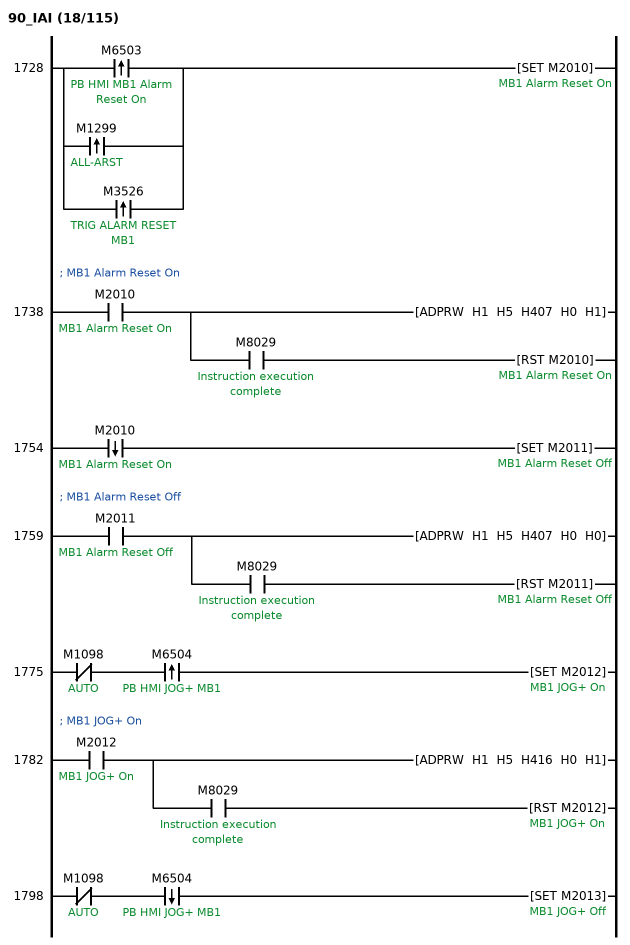
[picture p120: ladder of 90_IAI, rungs at steps 1728 to 1798]
1728  LDP     M6503  ; PB HMI MB1 Alarm Reset On
      ORP     M1299  ; ALL-ARST
      ORP     M3526  ; TRIG ALARM RESET MB1
      SET     M2010  ; MB1 Alarm Reset On
; MB1 Alarm Reset On
1738  LD      M2010  ; MB1 Alarm Reset On
      ADPRW   H1 H5 H407 H0 H1
      AND     M8029  ; Instruction execution complete
      RST     M2010  ; MB1 Alarm Reset On
1754  LDF     M2010  ; MB1 Alarm Reset On
      SET     M2011  ; MB1 Alarm Reset Off
; MB1 Alarm Reset Off
1759  LD      M2011  ; MB1 Alarm Reset Off
      ADPRW   H1 H5 H407 H0 H0
      AND     M8029  ; Instruction execution complete
      RST     M2011  ; MB1 Alarm Reset Off
1775  LDI     M1098  ; AUTO
      ANDP    M6504  ; PB HMI JOG+ MB1
      SET     M2012  ; MB1 JOG+ On
; MB1 JOG+ On
1782  LD      M2012  ; MB1 JOG+ On
      ADPRW   H1 H5 H416 H0 H1
      AND     M8029  ; Instruction execution complete
      RST     M2012  ; MB1 JOG+ On
1798  LDI     M1098  ; AUTO
      ANDF    M6504  ; PB HMI JOG+ MB1
      SET     M2013  ; MB1 JOG+ Off
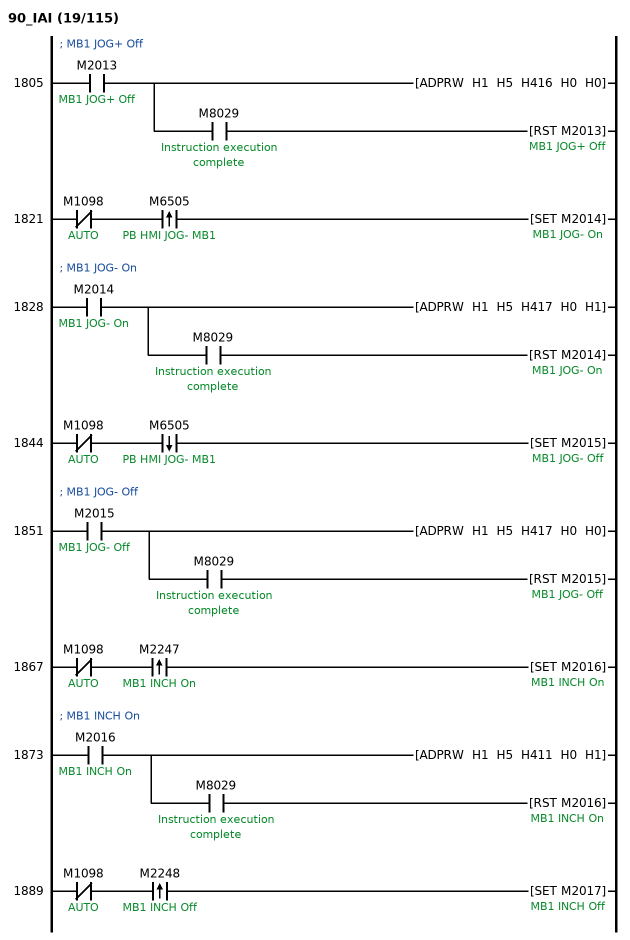
; MB1 JOG+ Off
1805  LD      M2013  ; MB1 JOG+ Off
      ADPRW   H1 H5 H416 H0 H0
      AND     M8029  ; Instruction execution complete
      RST     M2013  ; MB1 JOG+ Off
1821  LDI     M1098  ; AUTO
      ANDP    M6505  ; PB HMI JOG- MB1
      SET     M2014  ; MB1 JOG- On
; MB1 JOG- On
1828  LD      M2014  ; MB1 JOG- On
      ADPRW   H1 H5 H417 H0 H1
      AND     M8029  ; Instruction execution complete
      RST     M2014  ; MB1 JOG- On
1844  LDI     M1098  ; AUTO
      ANDF    M6505  ; PB HMI JOG- MB1
      SET     M2015  ; MB1 JOG- Off
; MB1 JOG- Off
1851  LD      M2015  ; MB1 JOG- Off
      ADPRW   H1 H5 H417 H0 H0
      AND     M8029  ; Instruction execution complete
      RST     M2015  ; MB1 JOG- Off
1867  LDI     M1098  ; AUTO
      ANDP    M2247  ; MB1 INCH On
      SET     M2016  ; MB1 INCH On
; MB1 INCH On
1873  LD      M2016  ; MB1 INCH On
      ADPRW   H1 H5 H411 H0 H1
      AND     M8029  ; Instruction execution complete
      RST     M2016  ; MB1 INCH On
1889  LDI     M1098  ; AUTO
      ANDP    M2248  ; MB1 INCH Off
      SET     M2017  ; MB1 INCH Off
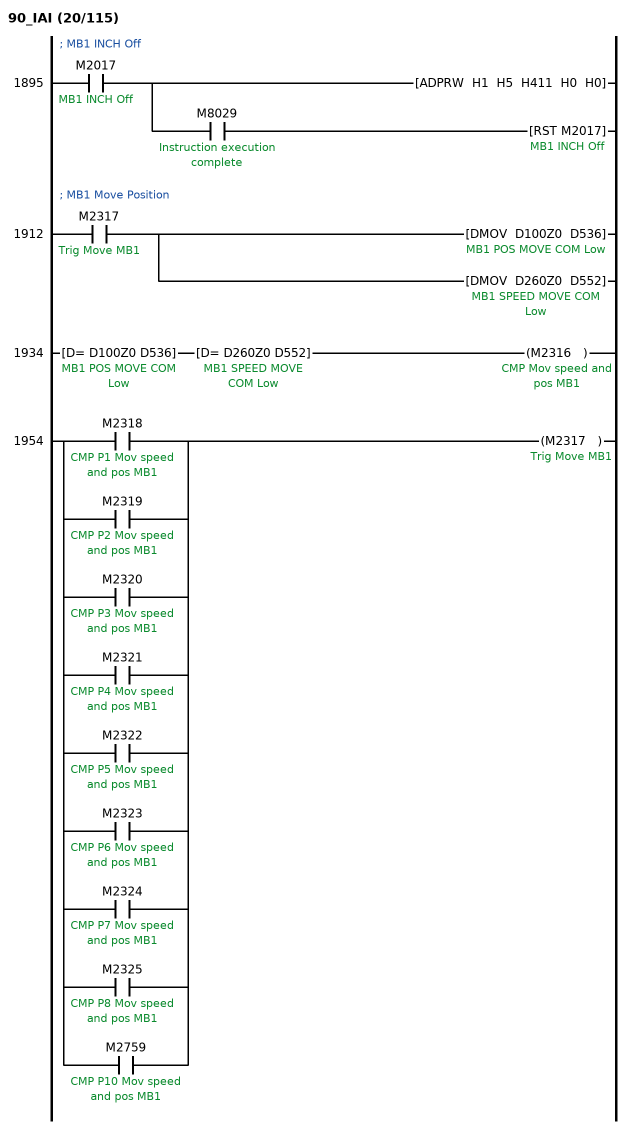
; MB1 INCH Off
1895  LD      M2017  ; MB1 INCH Off
      ADPRW   H1 H5 H411 H0 H0
      AND     M8029  ; Instruction execution complete
      RST     M2017  ; MB1 INCH Off
; MB1 Move Position
1912  LD      M2317  ; Trig Move MB1
      DMOV    D100Z0 D536
        [note] Position
      DMOV    D260Z0 D552
        [note] Speed
1934  LDD=    D100Z0 D536  ; MB1 POS MOVE COM Low
      ANDD=   D260Z0 D552  ; MB1 SPEED MOVE COM Low
      OUT     M2316  ; CMP Mov speed and pos MB1
1954  LD      M2318  ; CMP P1 Mov speed and pos MB1
      OR      M2319  ; CMP P2 Mov speed and pos MB1
      OR      M2320  ; CMP P3 Mov speed and pos MB1
      OR      M2321  ; CMP P4 Mov speed and pos MB1
      OR      M2322  ; CMP P5 Mov speed and pos MB1
      OR      M2323  ; CMP P6 Mov speed and pos MB1
      OR      M2324  ; CMP P7 Mov speed and pos MB1
      OR      M2325  ; CMP P8 Mov speed and pos MB1
      OR      M2759  ; CMP P10 Mov speed and pos MB1
      OUT     M2317  ; Trig Move MB1
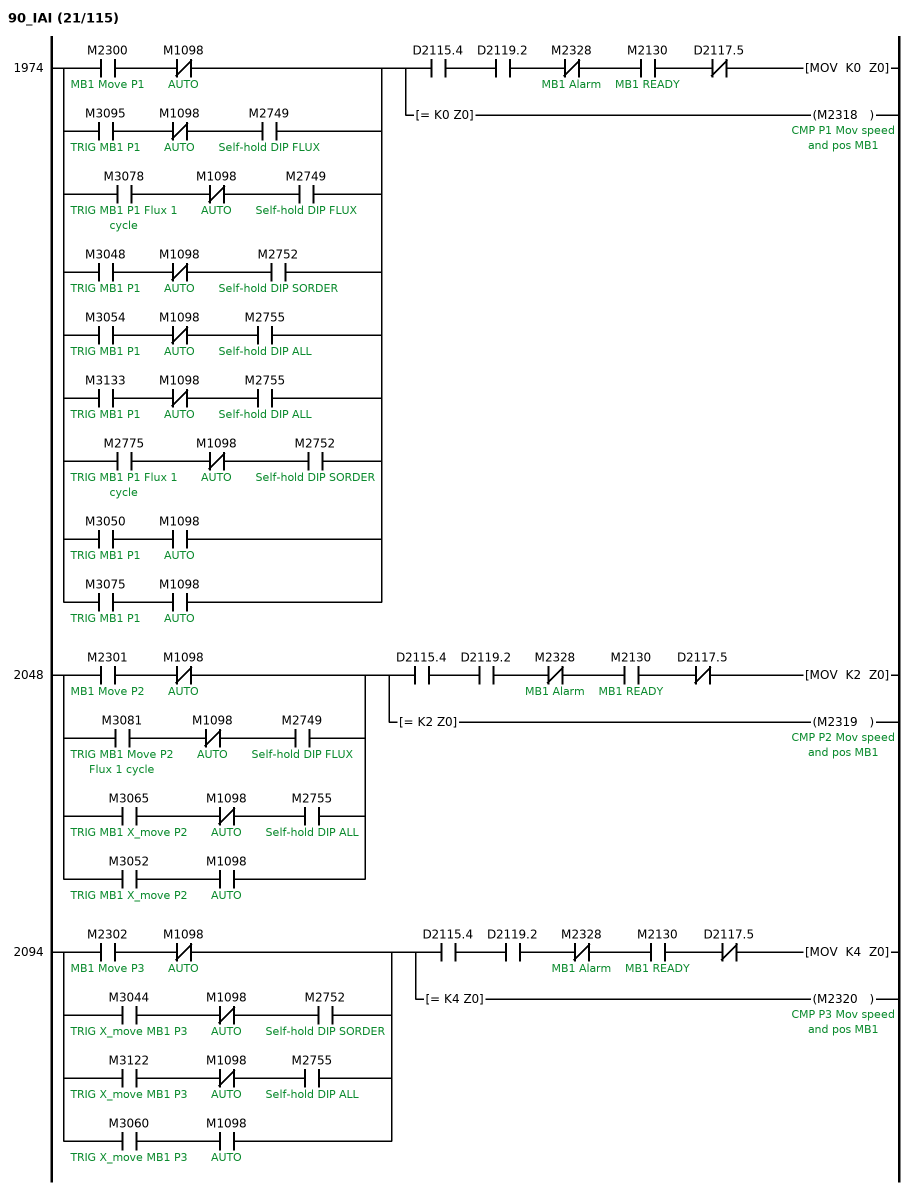
1974  LD      M2300  ; MB1 Move P1
      ANI     M1098  ; AUTO
      LD      M3095  ; TRIG MB1 P1
      ANI     M1098  ; AUTO
      AND     M2749  ; Self-hold DIP FLUX
      ORB
      LD      M3078  ; TRIG MB1 P1 Flux 1 cycle
      ANI     M1098  ; AUTO
      AND     M2749  ; Self-hold DIP FLUX
      ORB
      LD      M3048  ; TRIG MB1 P1
      ANI     M1098  ; AUTO
      AND     M2752  ; Self-hold DIP SORDER
      ORB
      LD      M3054  ; TRIG MB1 P1
      ANI     M1098  ; AUTO
      AND     M2755  ; Self-hold DIP ALL
      ORB
      LD      M3133  ; TRIG MB1 P1
      ANI     M1098  ; AUTO
      AND     M2755  ; Self-hold DIP ALL
      ORB
      LD      M2775  ; TRIG MB1 P1 Flux 1 cycle
      ANI     M1098  ; AUTO
      AND     M2752  ; Self-hold DIP SORDER
      ORB
      LD      M3050  ; TRIG MB1 P1
      AND     M1098  ; AUTO
      ORB
      LD      M3075  ; TRIG MB1 P1
      AND     M1098  ; AUTO
      ORB
      MPS
      AND     D2115.4
      AND     D2119.2
      ANI     M2328  ; MB1 Alarm
      AND     M2130  ; MB1 READY
      ANI     D2117.5
      MOV     K0 Z0
      MPP
      AND=    K0 Z0
      OUT     M2318  ; CMP P1 Mov speed and pos MB1
2048  LD      M2301  ; MB1 Move P2
      ANI     M1098  ; AUTO
      LD      M3081  ; TRIG MB1 Move P2 Flux 1 cycle
      ANI     M1098  ; AUTO
      AND     M2749  ; Self-hold DIP FLUX
      ORB
      LD      M3065  ; TRIG MB1 X_move P2
      ANI     M1098  ; AUTO
      AND     M2755  ; Self-hold DIP ALL
      ORB
      LD      M3052  ; TRIG MB1 X_move P2
      AND     M1098  ; AUTO
      ORB
      MPS
      AND     D2115.4
      AND     D2119.2
      ANI     M2328  ; MB1 Alarm
      AND     M2130  ; MB1 READY
      ANI     D2117.5
      MOV     K2 Z0
      MPP
      AND=    K2 Z0
      OUT     M2319  ; CMP P2 Mov speed and pos MB1
2094  LD      M2302  ; MB1 Move P3
      ANI     M1098  ; AUTO
      LD      M3044  ; TRIG X_move MB1 P3
      ANI     M1098  ; AUTO
      AND     M2752  ; Self-hold DIP SORDER
      ORB
      LD      M3122  ; TRIG X_move MB1 P3
      ANI     M1098  ; AUTO
      AND     M2755  ; Self-hold DIP ALL
      ORB
      LD      M3060  ; TRIG X_move MB1 P3
      AND     M1098  ; AUTO
      ORB
      MPS
      AND     D2115.4
      AND     D2119.2
      ANI     M2328  ; MB1 Alarm
      AND     M2130  ; MB1 READY
      ANI     D2117.5
      MOV     K4 Z0
      MPP
      AND=    K4 Z0
      OUT     M2320  ; CMP P3 Mov speed and pos MB1
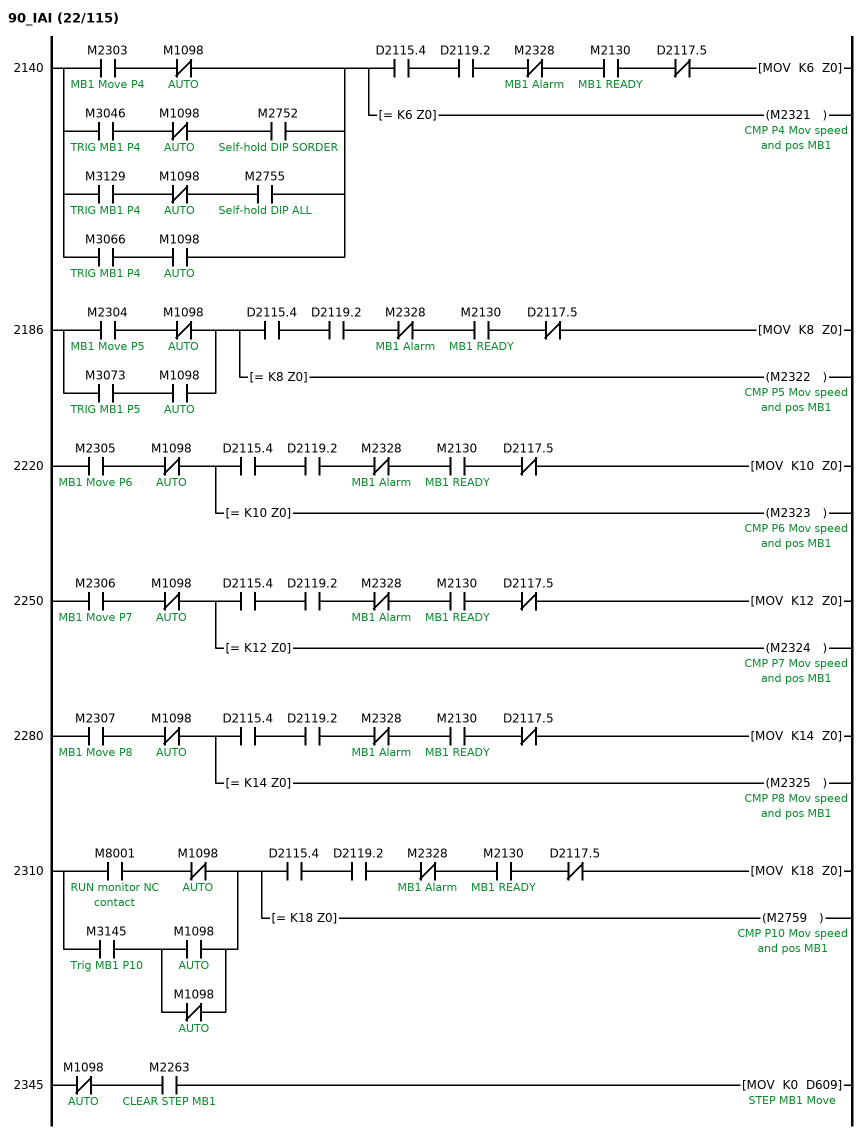
2140  LD      M2303  ; MB1 Move P4
      ANI     M1098  ; AUTO
      LD      M3046  ; TRIG MB1 P4
      ANI     M1098  ; AUTO
      AND     M2752  ; Self-hold DIP SORDER
      ORB
      LD      M3129  ; TRIG MB1 P4
      ANI     M1098  ; AUTO
      AND     M2755  ; Self-hold DIP ALL
      ORB
      LD      M3066  ; TRIG MB1 P4
      AND     M1098  ; AUTO
      ORB
      MPS
      AND     D2115.4
      AND     D2119.2
      ANI     M2328  ; MB1 Alarm
      AND     M2130  ; MB1 READY
      ANI     D2117.5
      MOV     K6 Z0
      MPP
      AND=    K6 Z0
      OUT     M2321  ; CMP P4 Mov speed and pos MB1
2186  LD      M2304  ; MB1 Move P5
      ANI     M1098  ; AUTO
      LD      M3073  ; TRIG MB1 P5
      AND     M1098  ; AUTO
      ORB
      MPS
      AND     D2115.4
      AND     D2119.2
      ANI     M2328  ; MB1 Alarm
      AND     M2130  ; MB1 READY
      ANI     D2117.5
      MOV     K8 Z0
      MPP
      AND=    K8 Z0
      OUT     M2322  ; CMP P5 Mov speed and pos MB1
2220  LD      M2305  ; MB1 Move P6
      ANI     M1098  ; AUTO
      MPS
      AND     D2115.4
      AND     D2119.2
      ANI     M2328  ; MB1 Alarm
      AND     M2130  ; MB1 READY
      ANI     D2117.5
      MOV     K10 Z0
      MPP
      AND=    K10 Z0
      OUT     M2323  ; CMP P6 Mov speed and pos MB1
2250  LD      M2306  ; MB1 Move P7
      ANI     M1098  ; AUTO
      MPS
      AND     D2115.4
      AND     D2119.2
      ANI     M2328  ; MB1 Alarm
      AND     M2130  ; MB1 READY
      ANI     D2117.5
      MOV     K12 Z0
      MPP
      AND=    K12 Z0
      OUT     M2324  ; CMP P7 Mov speed and pos MB1
2280  LD      M2307  ; MB1 Move P8
      ANI     M1098  ; AUTO
      MPS
      AND     D2115.4
      AND     D2119.2
      ANI     M2328  ; MB1 Alarm
      AND     M2130  ; MB1 READY
      ANI     D2117.5
      MOV     K14 Z0
      MPP
      AND=    K14 Z0
      OUT     M2325  ; CMP P8 Mov speed and pos MB1
2310  LD      M8001  ; RUN monitor NC contact
      ANI     M1098  ; AUTO
      LD      M3145  ; Trig MB1 P10
      LD      M1098  ; AUTO
      ORI     M1098  ; AUTO
      ANB
      ORB
      MPS
      AND     D2115.4
      AND     D2119.2
      ANI     M2328  ; MB1 Alarm
      AND     M2130  ; MB1 READY
      ANI     D2117.5
      MOV     K18 Z0
      MPP
      AND=    K18 Z0
      OUT     M2759  ; CMP P10 Mov speed and pos MB1
2345  LDI     M1098  ; AUTO
      AND     M2263  ; CLEAR STEP MB1
      MOV     K0 D609
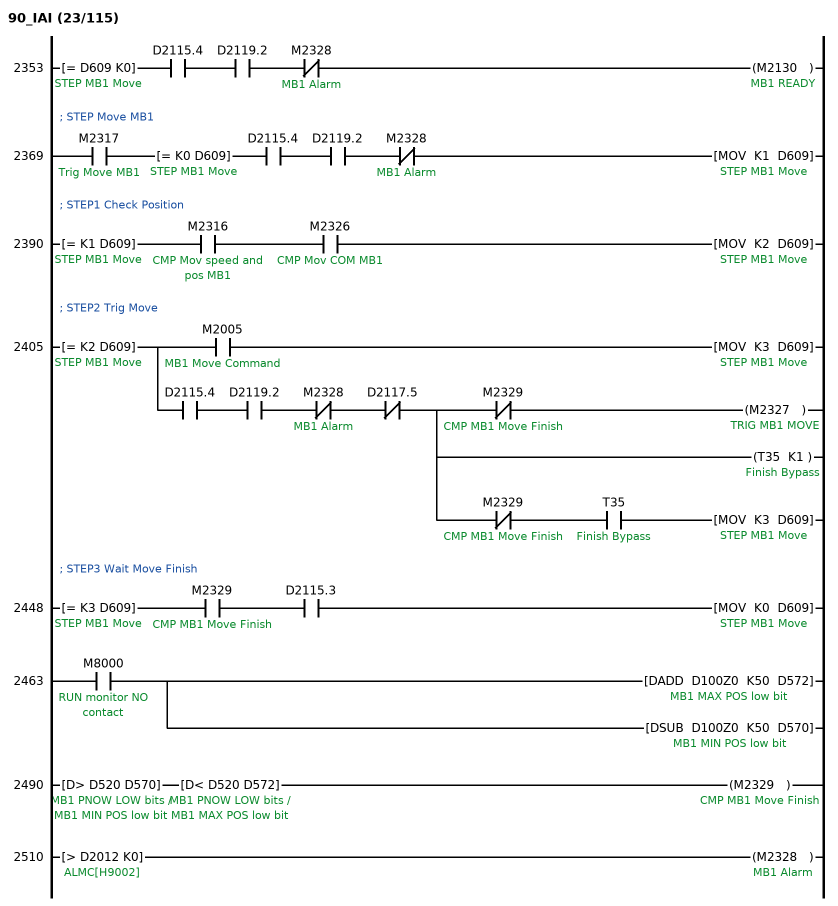
2353  LD=     D609 K0  ; STEP MB1 Move
      AND     D2115.4
      AND     D2119.2
      ANI     M2328  ; MB1 Alarm
      OUT     M2130  ; MB1 READY
; STEP Move MB1
2369  LD      M2317  ; Trig Move MB1
      AND=    K0 D609  ; STEP MB1 Move
      AND     D2115.4
      AND     D2119.2
      ANI     M2328  ; MB1 Alarm
      MOV     K1 D609
; STEP1 Check Position
2390  LD=     K1 D609  ; STEP MB1 Move
      AND     M2316  ; CMP Mov speed and pos MB1
      AND     M2326  ; CMP Mov COM MB1
      MOV     K2 D609
; STEP2 Trig Move
2405  LD=     K2 D609  ; STEP MB1 Move
      MPS
      AND     M2005  ; MB1 Move Command
      MOV     K3 D609
      MPP
      AND     D2115.4
      AND     D2119.2
      ANI     M2328  ; MB1 Alarm
      ANI     D2117.5
      MPS
      ANI     M2329  ; CMP MB1 Move Finish
      OUT     M2327  ; TRIG MB1 MOVE
      MPP
      OUT     T35 K1  ; Finish Bypass
      ANI     M2329  ; CMP MB1 Move Finish
      AND     T35  ; Finish Bypass
      MOV     K3 D609
; STEP3 Wait Move Finish
2448  LD=     K3 D609  ; STEP MB1 Move
      AND     M2329  ; CMP MB1 Move Finish
      AND     D2115.3
      MOV     K0 D609
2463  LD      M8000  ; RUN monitor NO contact
      DADD    D100Z0 K50 D572  ; MB1 MAX POS low bit
      DSUB    D100Z0 K50 D570  ; MB1 MIN POS low bit
2490  LDD>    D520 D570  ; MB1 PNOW LOW bits / MB1 MIN POS low bit
      ANDD<   D520 D572  ; MB1 PNOW LOW bits / MB1 MAX POS low bit
      OUT     M2329  ; CMP MB1 Move Finish
2510  LD>     D2012 K0  ; ALMC[H9002]
      OUT     M2328  ; MB1 Alarm
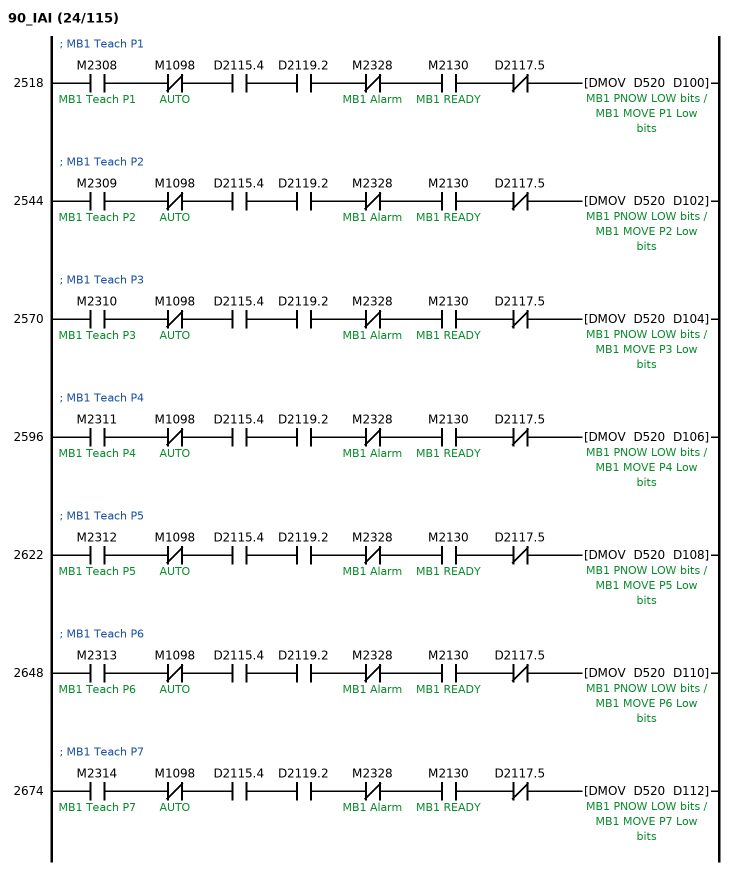
; MB1 Teach P1
2518  LD      M2308  ; MB1 Teach P1
      ANI     M1098  ; AUTO
      AND     D2115.4
      AND     D2119.2
      ANI     M2328  ; MB1 Alarm
      AND     M2130  ; MB1 READY
      ANI     D2117.5
      DMOV    D520 D100  ; MB1 MOVE P1 Low bits
; MB1 Teach P2
2544  LD      M2309  ; MB1 Teach P2
      ANI     M1098  ; AUTO
      AND     D2115.4
      AND     D2119.2
      ANI     M2328  ; MB1 Alarm
      AND     M2130  ; MB1 READY
      ANI     D2117.5
      DMOV    D520 D102  ; MB1 MOVE P2 Low bits
; MB1 Teach P3
2570  LD      M2310  ; MB1 Teach P3
      ANI     M1098  ; AUTO
      AND     D2115.4
      AND     D2119.2
      ANI     M2328  ; MB1 Alarm
      AND     M2130  ; MB1 READY
      ANI     D2117.5
      DMOV    D520 D104  ; MB1 MOVE P3 Low bits
; MB1 Teach P4
2596  LD      M2311  ; MB1 Teach P4
      ANI     M1098  ; AUTO
      AND     D2115.4
      AND     D2119.2
      ANI     M2328  ; MB1 Alarm
      AND     M2130  ; MB1 READY
      ANI     D2117.5
      DMOV    D520 D106  ; MB1 MOVE P4 Low bits
; MB1 Teach P5
2622  LD      M2312  ; MB1 Teach P5
      ANI     M1098  ; AUTO
      AND     D2115.4
      AND     D2119.2
      ANI     M2328  ; MB1 Alarm
      AND     M2130  ; MB1 READY
      ANI     D2117.5
      DMOV    D520 D108  ; MB1 MOVE P5 Low bits
; MB1 Teach P6
2648  LD      M2313  ; MB1 Teach P6
      ANI     M1098  ; AUTO
      AND     D2115.4
      AND     D2119.2
      ANI     M2328  ; MB1 Alarm
      AND     M2130  ; MB1 READY
      ANI     D2117.5
      DMOV    D520 D110  ; MB1 MOVE P6 Low bits
; MB1 Teach P7
2674  LD      M2314  ; MB1 Teach P7
      ANI     M1098  ; AUTO
      AND     D2115.4
      AND     D2119.2
      ANI     M2328  ; MB1 Alarm
      AND     M2130  ; MB1 READY
      ANI     D2117.5
      DMOV    D520 D112  ; MB1 MOVE P7 Low bits
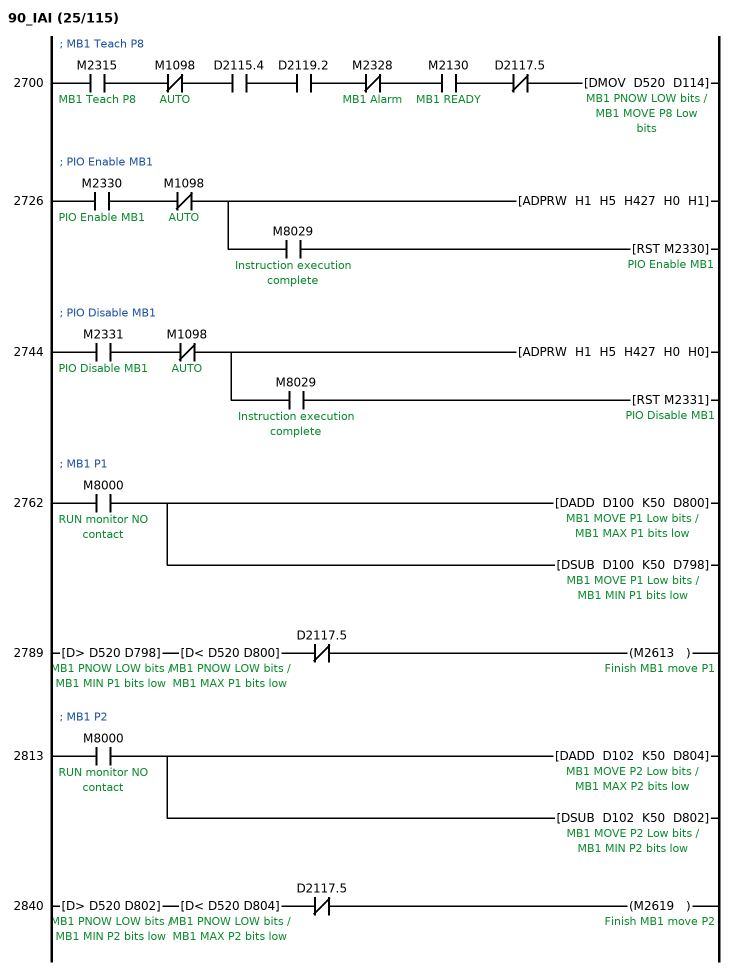
; MB1 Teach P8
2700  LD      M2315  ; MB1 Teach P8
      ANI     M1098  ; AUTO
      AND     D2115.4
      AND     D2119.2
      ANI     M2328  ; MB1 Alarm
      AND     M2130  ; MB1 READY
      ANI     D2117.5
      DMOV    D520 D114  ; MB1 MOVE P8 Low bits
; PIO Enable MB1
2726  LD      M2330  ; PIO Enable MB1
      ANI     M1098  ; AUTO
      ADPRW   H1 H5 H427 H0 H1
      AND     M8029  ; Instruction execution complete
      RST     M2330  ; PIO Enable MB1
; PIO Disable MB1
2744  LD      M2331  ; PIO Disable MB1
      ANI     M1098  ; AUTO
      ADPRW   H1 H5 H427 H0 H0
      AND     M8029  ; Instruction execution complete
      RST     M2331  ; PIO Disable MB1
; MB1 P1
2762  LD      M8000  ; RUN monitor NO contact
      DADD    D100 K50 D800  ; MB1 MAX P1 bits low
      DSUB    D100 K50 D798  ; MB1 MIN P1 bits low
2789  LDD>    D520 D798  ; MB1 PNOW LOW bits / MB1 MIN P1 bits low
      ANDD<   D520 D800  ; MB1 PNOW LOW bits / MB1 MAX P1 bits low
      ANI     D2117.5
      OUT     M2613  ; Finish MB1 move P1
; MB1 P2
2813  LD      M8000  ; RUN monitor NO contact
      DADD    D102 K50 D804  ; MB1 MAX P2 bits low
      DSUB    D102 K50 D802  ; MB1 MIN P2 bits low
2840  LDD>    D520 D802  ; MB1 PNOW LOW bits / MB1 MIN P2 bits low
      ANDD<   D520 D804  ; MB1 PNOW LOW bits / MB1 MAX P2 bits low
      ANI     D2117.5
      OUT     M2619  ; Finish MB1 move P2
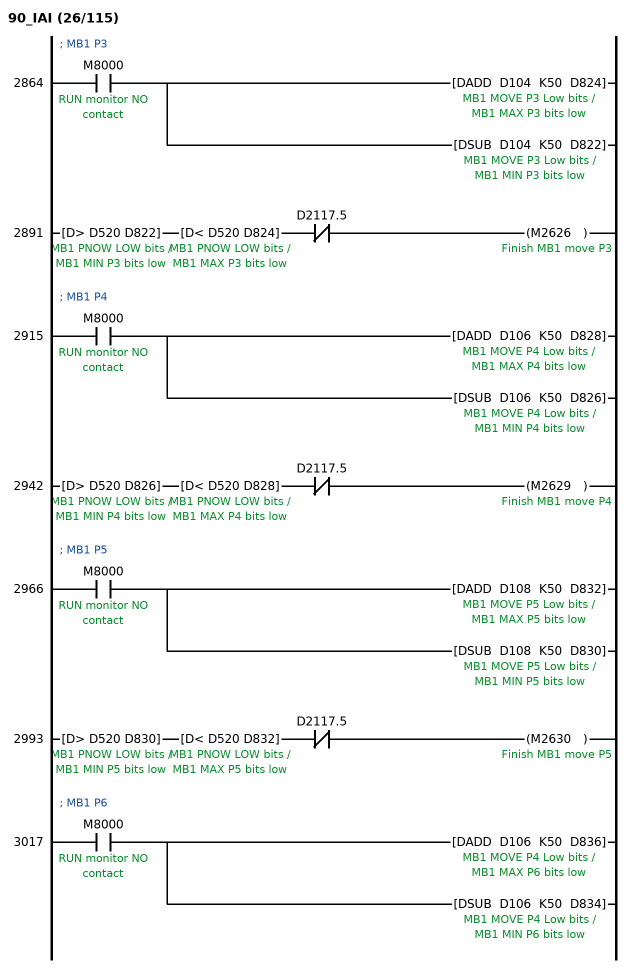
; MB1 P3
2864  LD      M8000  ; RUN monitor NO contact
      DADD    D104 K50 D824  ; MB1 MAX P3 bits low
      DSUB    D104 K50 D822  ; MB1 MIN P3 bits low
2891  LDD>    D520 D822  ; MB1 PNOW LOW bits / MB1 MIN P3 bits low
      ANDD<   D520 D824  ; MB1 PNOW LOW bits / MB1 MAX P3 bits low
      ANI     D2117.5
      OUT     M2626  ; Finish MB1 move P3
; MB1 P4
2915  LD      M8000  ; RUN monitor NO contact
      DADD    D106 K50 D828  ; MB1 MAX P4 bits low
      DSUB    D106 K50 D826  ; MB1 MIN P4 bits low
2942  LDD>    D520 D826  ; MB1 PNOW LOW bits / MB1 MIN P4 bits low
      ANDD<   D520 D828  ; MB1 PNOW LOW bits / MB1 MAX P4 bits low
      ANI     D2117.5
      OUT     M2629  ; Finish MB1 move P4
; MB1 P5
2966  LD      M8000  ; RUN monitor NO contact
      DADD    D108 K50 D832  ; MB1 MAX P5 bits low
      DSUB    D108 K50 D830  ; MB1 MIN P5 bits low
2993  LDD>    D520 D830  ; MB1 PNOW LOW bits / MB1 MIN P5 bits low
      ANDD<   D520 D832  ; MB1 PNOW LOW bits / MB1 MAX P5 bits low
      ANI     D2117.5
      OUT     M2630  ; Finish MB1 move P5
; MB1 P6
3017  LD      M8000  ; RUN monitor NO contact
      DADD    D106 K50 D836  ; MB1 MAX P6 bits low
      DSUB    D106 K50 D834  ; MB1 MIN P6 bits low
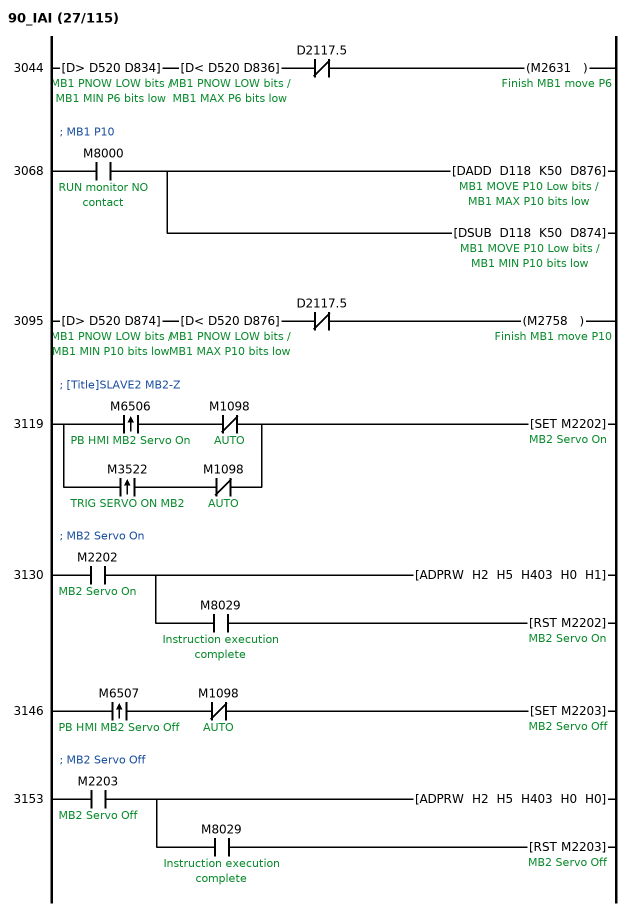
3044  LDD>    D520 D834  ; MB1 PNOW LOW bits / MB1 MIN P6 bits low
      ANDD<   D520 D836  ; MB1 PNOW LOW bits / MB1 MAX P6 bits low
      ANI     D2117.5
      OUT     M2631  ; Finish MB1 move P6
; MB1 P10
3068  LD      M8000  ; RUN monitor NO contact
      DADD    D118 K50 D876  ; MB1 MOVE P10 Low bits / MB1 MAX P10 bits low
      DSUB    D118 K50 D874  ; MB1 MIN P10 bits low
3095  LDD>    D520 D874  ; MB1 PNOW LOW bits / MB1 MIN P10 bits low
      ANDD<   D520 D876  ; MB1 PNOW LOW bits / MB1 MAX P10 bits low
      ANI     D2117.5
      OUT     M2758  ; Finish MB1 move P10
; [Title]SLAVE2 MB2-Z
3119  LDP     M6506  ; PB HMI MB2 Servo On
      ANI     M1098  ; AUTO
      LDP     M3522  ; TRIG SERVO ON MB2
      ANI     M1098  ; AUTO
      ORB
      SET     M2202  ; MB2 Servo On
; MB2 Servo On
3130  LD      M2202  ; MB2 Servo On
      ADPRW   H2 H5 H403 H0 H1
      AND     M8029  ; Instruction execution complete
      RST     M2202  ; MB2 Servo On
3146  LDP     M6507  ; PB HMI MB2 Servo Off
      ANI     M1098  ; AUTO
      SET     M2203  ; MB2 Servo Off
; MB2 Servo Off
3153  LD      M2203  ; MB2 Servo Off
      ADPRW   H2 H5 H403 H0 H0
      AND     M8029  ; Instruction execution complete
      RST     M2203  ; MB2 Servo Off
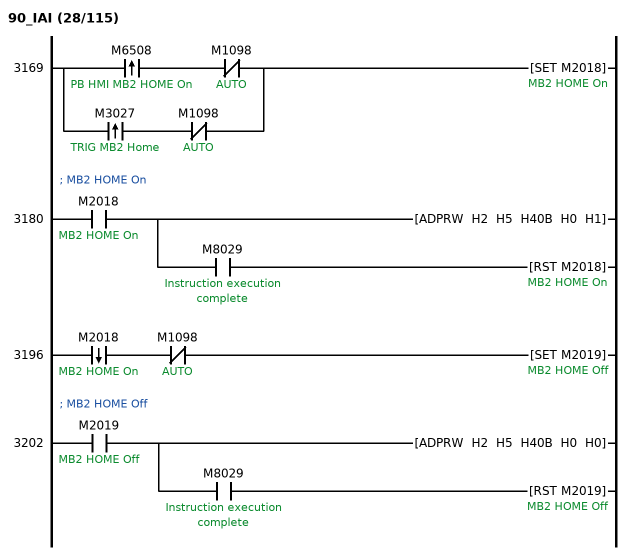
3169  LDP     M6508  ; PB HMI MB2 HOME On
      ANI     M1098  ; AUTO
      LDP     M3027  ; TRIG MB2 Home
      ANI     M1098  ; AUTO
      ORB
      SET     M2018  ; MB2 HOME On
; MB2 HOME On
3180  LD      M2018  ; MB2 HOME On
      ADPRW   H2 H5 H40B H0 H1
      AND     M8029  ; Instruction execution complete
      RST     M2018  ; MB2 HOME On
3196  LDF     M2018  ; MB2 HOME On
      ANI     M1098  ; AUTO
      SET     M2019  ; MB2 HOME Off
; MB2 HOME Off
3202  LD      M2019  ; MB2 HOME Off
      ADPRW   H2 H5 H40B H0 H0
      AND     M8029  ; Instruction execution complete
      RST     M2019  ; MB2 HOME Off
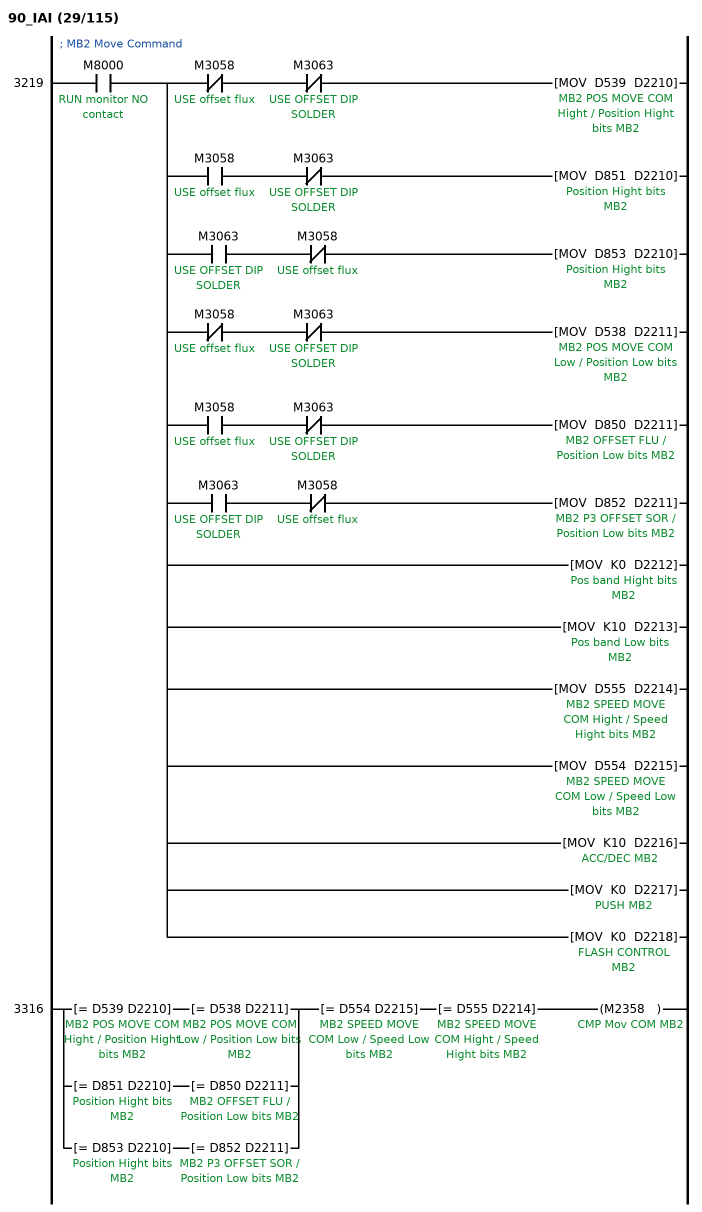
; MB2 Move Command
3219  LD      M8000  ; RUN monitor NO contact
      MPS
      ANI     M3058  ; USE offset flux
      ANI     M3063  ; USE OFFSET DIP SOLDER
      MOV     D539 D2210  ; MB2 POS MOVE COM Hight / Position Hight bits MB2
      MRD
      AND     M3058  ; USE offset flux
      ANI     M3063  ; USE OFFSET DIP SOLDER
      MOV     D851 D2210
      MRD
      AND     M3063  ; USE OFFSET DIP SOLDER
      ANI     M3058  ; USE offset flux
      MOV     D853 D2210
      MRD
      ANI     M3058  ; USE offset flux
      ANI     M3063  ; USE OFFSET DIP SOLDER
      MOV     D538 D2211  ; MB2 POS MOVE COM Low / Position Low bits MB2
      MRD
      AND     M3058  ; USE offset flux
      ANI     M3063  ; USE OFFSET DIP SOLDER
      MOV     D850 D2211  ; MB2 OFFSET FLU
      MRD
      AND     M3063  ; USE OFFSET DIP SOLDER
      ANI     M3058  ; USE offset flux
      MOV     D852 D2211  ; MB2 P3 OFFSET SOR
      MPP
      MOV     K0 D2212  ; Pos band Hight bits MB2
      MOV     K10 D2213  ; Pos band Low bits MB2
      MOV     D555 D2214  ; MB2 SPEED MOVE COM Hight / Speed Hight bits MB2
      MOV     D554 D2215  ; MB2 SPEED MOVE COM Low / Speed Low bits MB2
      MOV     K10 D2216  ; ACC/DEC MB2
      MOV     K0 D2217  ; PUSH MB2
      MOV     K0 D2218  ; FLASH CONTROL MB2
3316  LD=     D539 D2210  ; MB2 POS MOVE COM Hight / Position Hight bits MB2
      AND=    D538 D2211  ; MB2 POS MOVE COM Low / Position Low bits MB2
      LD=     D851 D2210  ; Position Hight bits MB2
      AND=    D850 D2211  ; MB2 OFFSET FLU / Position Low bits MB2
      ORB
      LD=     D853 D2210  ; Position Hight bits MB2
      AND=    D852 D2211  ; MB2 P3 OFFSET SOR / Position Low bits MB2
      ORB
      AND=    D554 D2215  ; MB2 SPEED MOVE COM Low / Speed Low bits MB2
      AND=    D555 D2214  ; MB2 SPEED MOVE COM Hight / Speed Hight bits MB2
      OUT     M2358  ; CMP Mov COM MB2
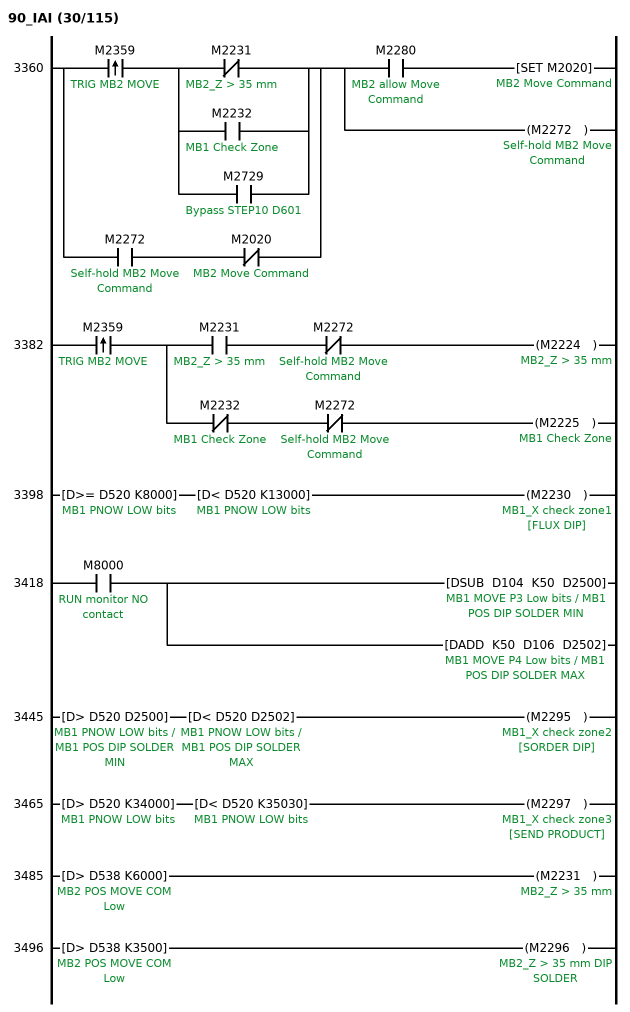
3360  LDP     M2359  ; TRIG MB2 MOVE
      LDI     M2231  ; MB2_Z > 35 mm
      OR      M2232  ; MB1 Check Zone
      OR      M2729  ; Bypass STEP10 D601
      ANB
      LD      M2272  ; Self-hold MB2 Move Command
      ANI     M2020  ; MB2 Move Command
      ORB
      MPS
      AND     M2280  ; MB2 allow Move Command
      SET     M2020  ; MB2 Move Command
      MPP
      OUT     M2272  ; Self-hold MB2 Move Command
3382  LDP     M2359  ; TRIG MB2 MOVE
      MPS
      AND     M2231  ; MB2_Z > 35 mm
      ANI     M2272  ; Self-hold MB2 Move Command
      OUT     M2224  ; MB2_Z > 35 mm
      MPP
      ANI     M2232  ; MB1 Check Zone
      ANI     M2272  ; Self-hold MB2 Move Command
      OUT     M2225  ; MB1 Check Zone
3398  LDD>=   D520 K8000  ; MB1 PNOW LOW bits
      ANDD<   D520 K13000  ; MB1 PNOW LOW bits
      OUT     M2230  ; MB1_X check zone1 [FLUX DIP]
3418  LD      M8000  ; RUN monitor NO contact
      DSUB    D104 K50 D2500  ; MB1 POS DIP SOLDER MIN
      DADD    K50 D106 D2502  ; MB1 POS DIP SOLDER MAX
3445  LDD>    D520 D2500  ; MB1 PNOW LOW bits / MB1 POS DIP SOLDER MIN
      ANDD<   D520 D2502  ; MB1 PNOW LOW bits / MB1 POS DIP SOLDER MAX
      OUT     M2295  ; MB1_X check zone2 [SORDER DIP]
3465  LDD>    D520 K34000  ; MB1 PNOW LOW bits
      ANDD<   D520 K35030  ; MB1 PNOW LOW bits
      OUT     M2297  ; MB1_X check zone3 [SEND PRODUCT]
3485  LDD>    D538 K6000  ; MB2 POS MOVE COM Low
      OUT     M2231  ; MB2_Z > 35 mm
3496  LDD>    D538 K3500  ; MB2 POS MOVE COM Low
      OUT     M2296  ; MB2_Z > 35 mm DIP SOLDER
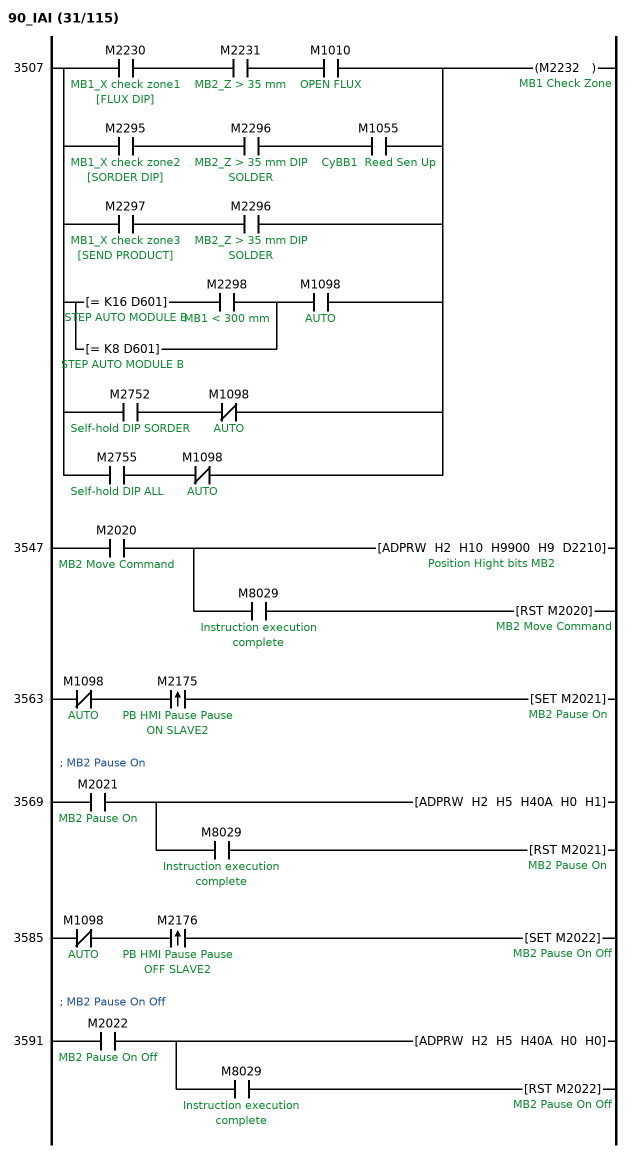
3507  LD      M2230  ; MB1_X check zone1 [FLUX DIP]
      AND     M2231  ; MB2_Z > 35 mm
      AND     M1010  ; OPEN FLUX
      LD      M2295  ; MB1_X check zone2 [SORDER DIP]
      AND     M2296  ; MB2_Z > 35 mm DIP SOLDER
      AND     M1055  ; CyBB1  Reed Sen Up
      ORB
      LD      M2297  ; MB1_X check zone3 [SEND PRODUCT]
      AND     M2296  ; MB2_Z > 35 mm DIP SOLDER
      ORB
      LD=     K16 D601  ; STEP AUTO MODULE B
      AND     M2298  ; MB1 < 300 mm
      OR=     K8 D601  ; STEP AUTO MODULE B
      AND     M1098  ; AUTO
      ORB
      LD      M2752  ; Self-hold DIP SORDER
      ANI     M1098  ; AUTO
      ORB
      LD      M2755  ; Self-hold DIP ALL
      ANI     M1098  ; AUTO
      ORB
      OUT     M2232  ; MB1 Check Zone
3547  LD      M2020  ; MB2 Move Command
      ADPRW   H2 H10 H9900 H9 D2210
      AND     M8029  ; Instruction execution complete
      RST     M2020  ; MB2 Move Command
3563  LDI     M1098  ; AUTO
      ANDP    M2175  ; PB HMI Pause Pause ON SLAVE2
      SET     M2021  ; MB2 Pause On
; MB2 Pause On
3569  LD      M2021  ; MB2 Pause On
      ADPRW   H2 H5 H40A H0 H1
      AND     M8029  ; Instruction execution complete
      RST     M2021  ; MB2 Pause On
3585  LDI     M1098  ; AUTO
      ANDP    M2176  ; PB HMI Pause Pause OFF SLAVE2
      SET     M2022  ; MB2 Pause On Off
; MB2 Pause On Off
3591  LD      M2022  ; MB2 Pause On Off
      ADPRW   H2 H5 H40A H0 H0
      AND     M8029  ; Instruction execution complete
      RST     M2022  ; MB2 Pause On Off
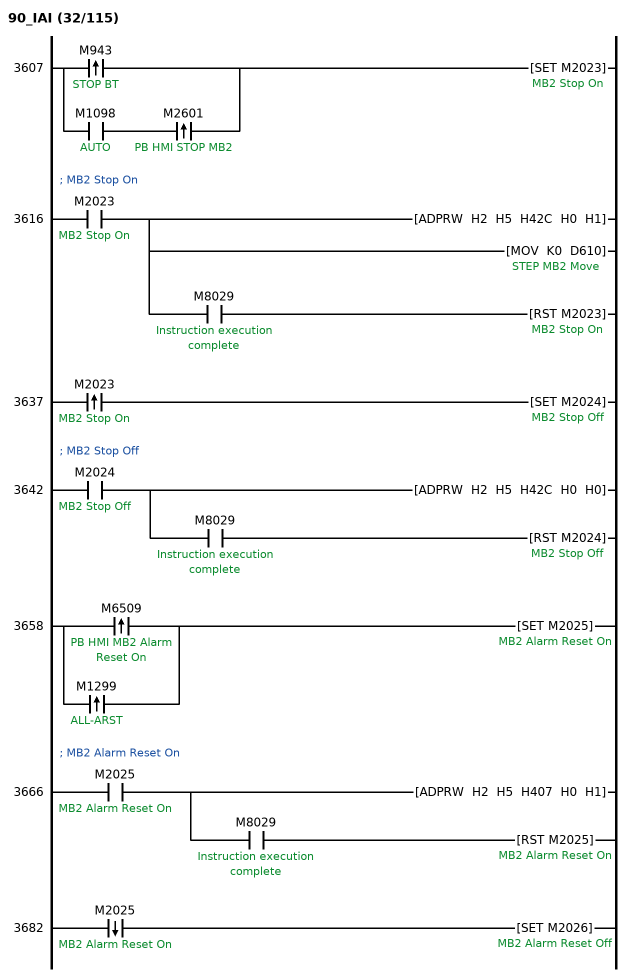
3607  LDP     M943  ; STOP BT
      LD      M1098  ; AUTO
      ANDP    M2601  ; PB HMI STOP MB2
      ORB
      SET     M2023  ; MB2 Stop On
; MB2 Stop On
3616  LD      M2023  ; MB2 Stop On
      ADPRW   H2 H5 H42C H0 H1
      MOV     K0 D610  ; STEP MB2 Move
      AND     M8029  ; Instruction execution complete
      RST     M2023  ; MB2 Stop On
3637  LDP     M2023  ; MB2 Stop On
      SET     M2024  ; MB2 Stop Off
; MB2 Stop Off
3642  LD      M2024  ; MB2 Stop Off
      ADPRW   H2 H5 H42C H0 H0
      AND     M8029  ; Instruction execution complete
      RST     M2024  ; MB2 Stop Off
3658  LDP     M6509  ; PB HMI MB2 Alarm Reset On
      ORP     M1299  ; ALL-ARST
      SET     M2025  ; MB2 Alarm Reset On
; MB2 Alarm Reset On
3666  LD      M2025  ; MB2 Alarm Reset On
      ADPRW   H2 H5 H407 H0 H1
      AND     M8029  ; Instruction execution complete
      RST     M2025  ; MB2 Alarm Reset On
3682  LDF     M2025  ; MB2 Alarm Reset On
      SET     M2026  ; MB2 Alarm Reset Off
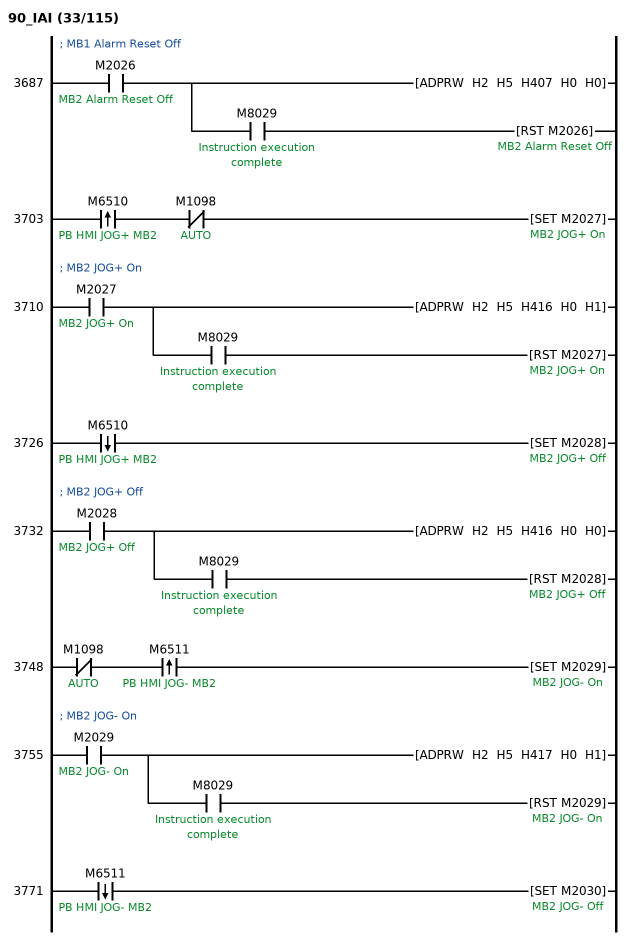
; MB1 Alarm Reset Off
3687  LD      M2026  ; MB2 Alarm Reset Off
      ADPRW   H2 H5 H407 H0 H0
      AND     M8029  ; Instruction execution complete
      RST     M2026  ; MB2 Alarm Reset Off
3703  LDP     M6510  ; PB HMI JOG+ MB2
      ANI     M1098  ; AUTO
      SET     M2027  ; MB2 JOG+ On
; MB2 JOG+ On
3710  LD      M2027  ; MB2 JOG+ On
      ADPRW   H2 H5 H416 H0 H1
      AND     M8029  ; Instruction execution complete
      RST     M2027  ; MB2 JOG+ On
3726  LDF     M6510  ; PB HMI JOG+ MB2
      SET     M2028  ; MB2 JOG+ Off
; MB2 JOG+ Off
3732  LD      M2028  ; MB2 JOG+ Off
      ADPRW   H2 H5 H416 H0 H0
      AND     M8029  ; Instruction execution complete
      RST     M2028  ; MB2 JOG+ Off
3748  LDI     M1098  ; AUTO
      ANDP    M6511  ; PB HMI JOG- MB2
      SET     M2029  ; MB2 JOG- On
; MB2 JOG- On
3755  LD      M2029  ; MB2 JOG- On
      ADPRW   H2 H5 H417 H0 H1
      AND     M8029  ; Instruction execution complete
      RST     M2029  ; MB2 JOG- On
3771  LDF     M6511  ; PB HMI JOG- MB2
      SET     M2030  ; MB2 JOG- Off
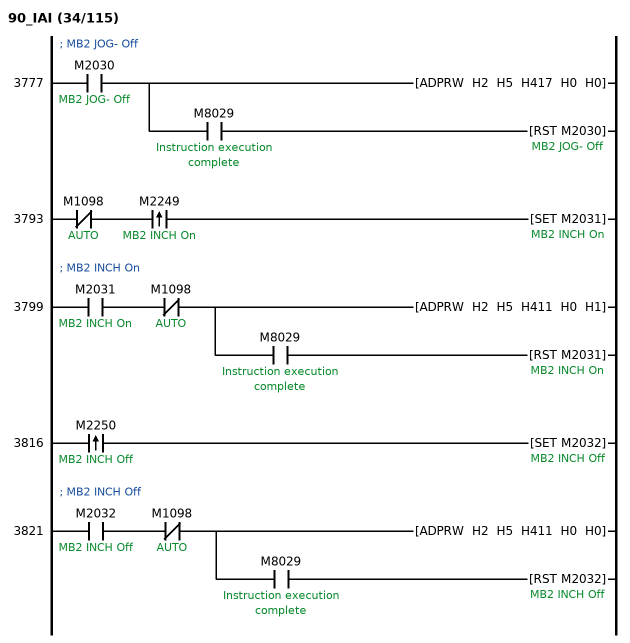
; MB2 JOG- Off
3777  LD      M2030  ; MB2 JOG- Off
      ADPRW   H2 H5 H417 H0 H0
      AND     M8029  ; Instruction execution complete
      RST     M2030  ; MB2 JOG- Off
3793  LDI     M1098  ; AUTO
      ANDP    M2249  ; MB2 INCH On
      SET     M2031  ; MB2 INCH On
; MB2 INCH On
3799  LD      M2031  ; MB2 INCH On
      ANI     M1098  ; AUTO
      ADPRW   H2 H5 H411 H0 H1
      AND     M8029  ; Instruction execution complete
      RST     M2031  ; MB2 INCH On
3816  LDP     M2250  ; MB2 INCH Off
      SET     M2032  ; MB2 INCH Off
; MB2 INCH Off
3821  LD      M2032  ; MB2 INCH Off
      ANI     M1098  ; AUTO
      ADPRW   H2 H5 H411 H0 H0
      AND     M8029  ; Instruction execution complete
      RST     M2032  ; MB2 INCH Off
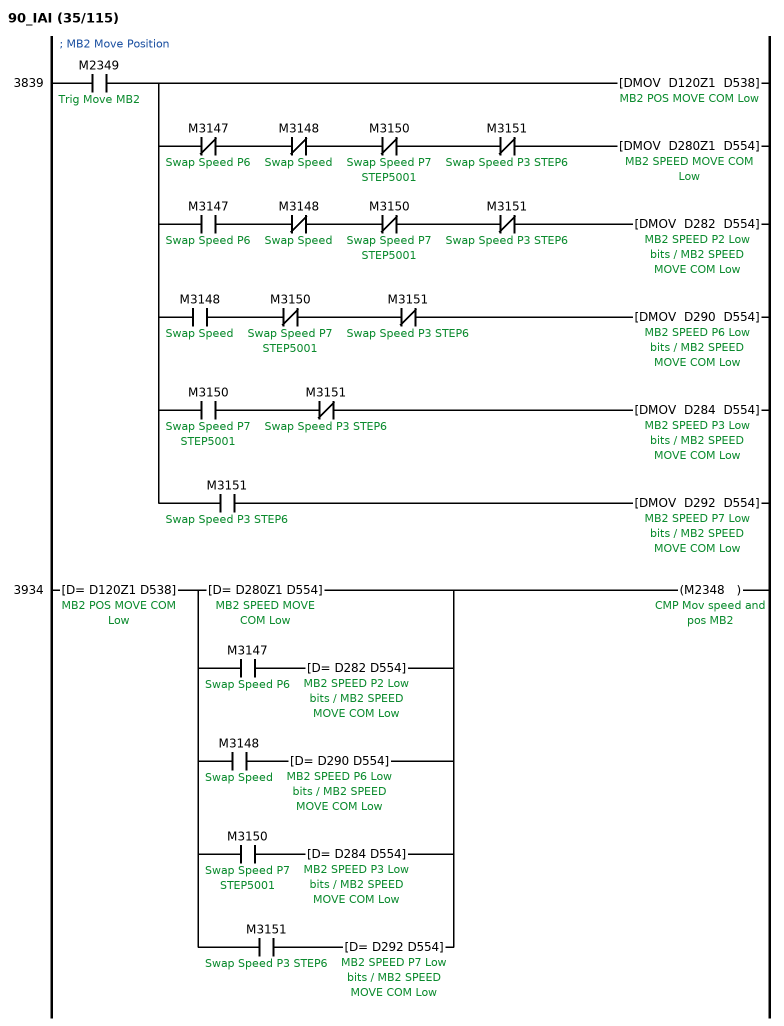
; MB2 Move Position
3839  LD      M2349  ; Trig Move MB2
      DMOV    D120Z1 D538
        [note] Position
      MPS
      ANI     M3147  ; Swap Speed P6
      ANI     M3148  ; Swap Speed
      ANI     M3150  ; Swap Speed P7 STEP5001
      ANI     M3151  ; Swap Speed P3 STEP6
      DMOV    D280Z1 D554
        [note] Speed
      MRD
      AND     M3147  ; Swap Speed P6
      ANI     M3148  ; Swap Speed
      ANI     M3150  ; Swap Speed P7 STEP5001
      ANI     M3151  ; Swap Speed P3 STEP6
      DMOV    D282 D554  ; MB2 SPEED P2 Low bits
        [note] Swap Speed
      MRD
      AND     M3148  ; Swap Speed
      ANI     M3150  ; Swap Speed P7 STEP5001
      ANI     M3151  ; Swap Speed P3 STEP6
      DMOV    D290 D554  ; MB2 SPEED P6 Low bits
        [note] Swap Speed
      MRD
      AND     M3150  ; Swap Speed P7 STEP5001
      ANI     M3151  ; Swap Speed P3 STEP6
      DMOV    D284 D554  ; MB2 SPEED P3 Low bits
        [note] Swap Speed
      MPP
      AND     M3151  ; Swap Speed P3 STEP6
      DMOV    D292 D554  ; MB2 SPEED P7 Low bits
        [note] Swap Speed
3934  LDD=    D120Z1 D538  ; MB2 POS MOVE COM Low
      LDD=    D280Z1 D554  ; MB2 SPEED MOVE COM Low
      LD      M3147  ; Swap Speed P6
      ANDD=   D282 D554  ; MB2 SPEED P2 Low bits / MB2 SPEED MOVE COM Low
      ORB
      LD      M3148  ; Swap Speed
      ANDD=   D290 D554  ; MB2 SPEED P6 Low bits / MB2 SPEED MOVE COM Low
      ORB
      LD      M3150  ; Swap Speed P7 STEP5001
      ANDD=   D284 D554  ; MB2 SPEED P3 Low bits / MB2 SPEED MOVE COM Low
      ORB
      LD      M3151  ; Swap Speed P3 STEP6
      ANDD=   D292 D554  ; MB2 SPEED P7 Low bits / MB2 SPEED MOVE COM Low
      ORB
      ANB
      OUT     M2348  ; CMP Mov speed and pos MB2
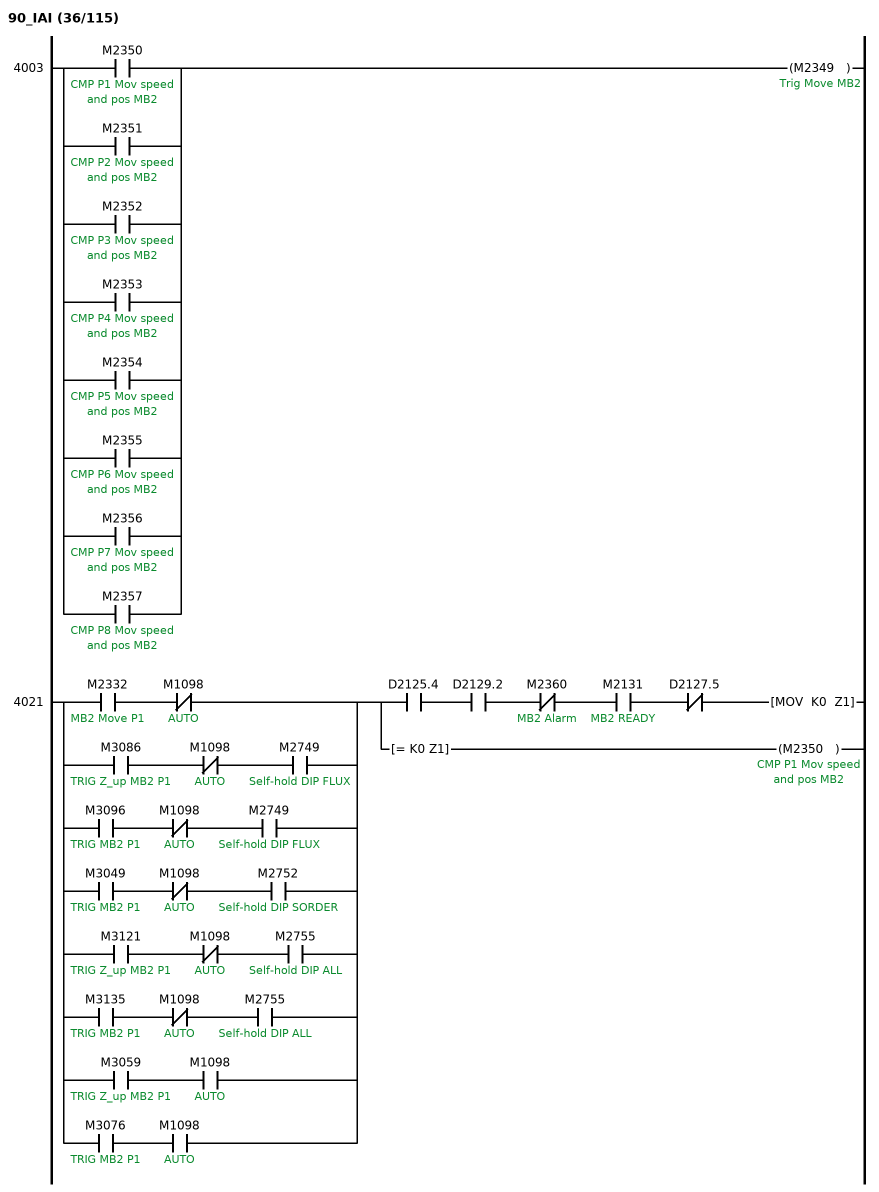
4003  LD      M2350  ; CMP P1 Mov speed and pos MB2
      OR      M2351  ; CMP P2 Mov speed and pos MB2
      OR      M2352  ; CMP P3 Mov speed and pos MB2
      OR      M2353  ; CMP P4 Mov speed and pos MB2
      OR      M2354  ; CMP P5 Mov speed and pos MB2
      OR      M2355  ; CMP P6 Mov speed and pos MB2
      OR      M2356  ; CMP P7 Mov speed and pos MB2
      OR      M2357  ; CMP P8 Mov speed and pos MB2
      OUT     M2349  ; Trig Move MB2
4021  LD      M2332  ; MB2 Move P1
      ANI     M1098  ; AUTO
      LD      M3086  ; TRIG Z_up MB2 P1
      ANI     M1098  ; AUTO
      AND     M2749  ; Self-hold DIP FLUX
      ORB
      LD      M3096  ; TRIG MB2 P1
      ANI     M1098  ; AUTO
      AND     M2749  ; Self-hold DIP FLUX
      ORB
      LD      M3049  ; TRIG MB2 P1
      ANI     M1098  ; AUTO
      AND     M2752  ; Self-hold DIP SORDER
      ORB
      LD      M3121  ; TRIG Z_up MB2 P1
      ANI     M1098  ; AUTO
      AND     M2755  ; Self-hold DIP ALL
      ORB
      LD      M3135  ; TRIG MB2 P1
      ANI     M1098  ; AUTO
      AND     M2755  ; Self-hold DIP ALL
      ORB
      LD      M3059  ; TRIG Z_up MB2 P1
      AND     M1098  ; AUTO
      ORB
      LD      M3076  ; TRIG MB2 P1
      AND     M1098  ; AUTO
      ORB
      MPS
      AND     D2125.4
      AND     D2129.2
      ANI     M2360  ; MB2 Alarm
      AND     M2131  ; MB2 READY
      ANI     D2127.5
      MOV     K0 Z1
      MPP
      AND=    K0 Z1
      OUT     M2350  ; CMP P1 Mov speed and pos MB2
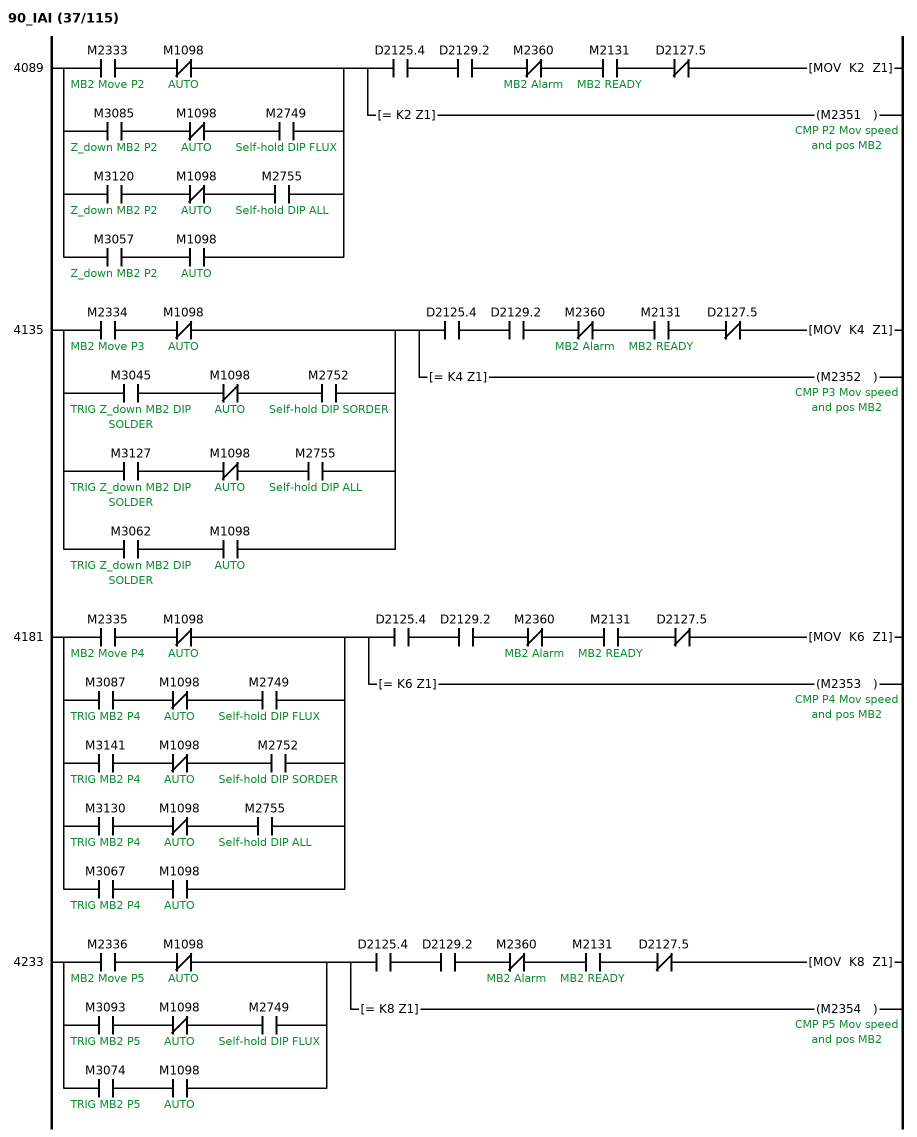
4089  LD      M2333  ; MB2 Move P2
      ANI     M1098  ; AUTO
      LD      M3085  ; Z_down MB2 P2
      ANI     M1098  ; AUTO
      AND     M2749  ; Self-hold DIP FLUX
      ORB
      LD      M3120  ; Z_down MB2 P2
      ANI     M1098  ; AUTO
      AND     M2755  ; Self-hold DIP ALL
      ORB
      LD      M3057  ; Z_down MB2 P2
      AND     M1098  ; AUTO
      ORB
      MPS
      AND     D2125.4
      AND     D2129.2
      ANI     M2360  ; MB2 Alarm
      AND     M2131  ; MB2 READY
      ANI     D2127.5
      MOV     K2 Z1
      MPP
      AND=    K2 Z1
      OUT     M2351  ; CMP P2 Mov speed and pos MB2
4135  LD      M2334  ; MB2 Move P3
      ANI     M1098  ; AUTO
      LD      M3045  ; TRIG Z_down MB2 DIP SOLDER
      ANI     M1098  ; AUTO
      AND     M2752  ; Self-hold DIP SORDER
      ORB
      LD      M3127  ; TRIG Z_down MB2 DIP SOLDER
      ANI     M1098  ; AUTO
      AND     M2755  ; Self-hold DIP ALL
      ORB
      LD      M3062  ; TRIG Z_down MB2 DIP SOLDER
      AND     M1098  ; AUTO
      ORB
      MPS
      AND     D2125.4
      AND     D2129.2
      ANI     M2360  ; MB2 Alarm
      AND     M2131  ; MB2 READY
      ANI     D2127.5
      MOV     K4 Z1
      MPP
      AND=    K4 Z1
      OUT     M2352  ; CMP P3 Mov speed and pos MB2
4181  LD      M2335  ; MB2 Move P4
      ANI     M1098  ; AUTO
      LD      M3087  ; TRIG MB2 P4
      ANI     M1098  ; AUTO
      AND     M2749  ; Self-hold DIP FLUX
      ORB
      LD      M3141  ; TRIG MB2 P4
      ANI     M1098  ; AUTO
      AND     M2752  ; Self-hold DIP SORDER
      ORB
      LD      M3130  ; TRIG MB2 P4
      ANI     M1098  ; AUTO
      AND     M2755  ; Self-hold DIP ALL
      ORB
      LD      M3067  ; TRIG MB2 P4
      AND     M1098  ; AUTO
      ORB
      MPS
      AND     D2125.4
      AND     D2129.2
      ANI     M2360  ; MB2 Alarm
      AND     M2131  ; MB2 READY
      ANI     D2127.5
      MOV     K6 Z1
      MPP
      AND=    K6 Z1
      OUT     M2353  ; CMP P4 Mov speed and pos MB2
4233  LD      M2336  ; MB2 Move P5
      ANI     M1098  ; AUTO
      LD      M3093  ; TRIG MB2 P5
      ANI     M1098  ; AUTO
      AND     M2749  ; Self-hold DIP FLUX
      ORB
      LD      M3074  ; TRIG MB2 P5
      AND     M1098  ; AUTO
      ORB
      MPS
      AND     D2125.4
      AND     D2129.2
      ANI     M2360  ; MB2 Alarm
      AND     M2131  ; MB2 READY
      ANI     D2127.5
      MOV     K8 Z1
      MPP
      AND=    K8 Z1
      OUT     M2354  ; CMP P5 Mov speed and pos MB2
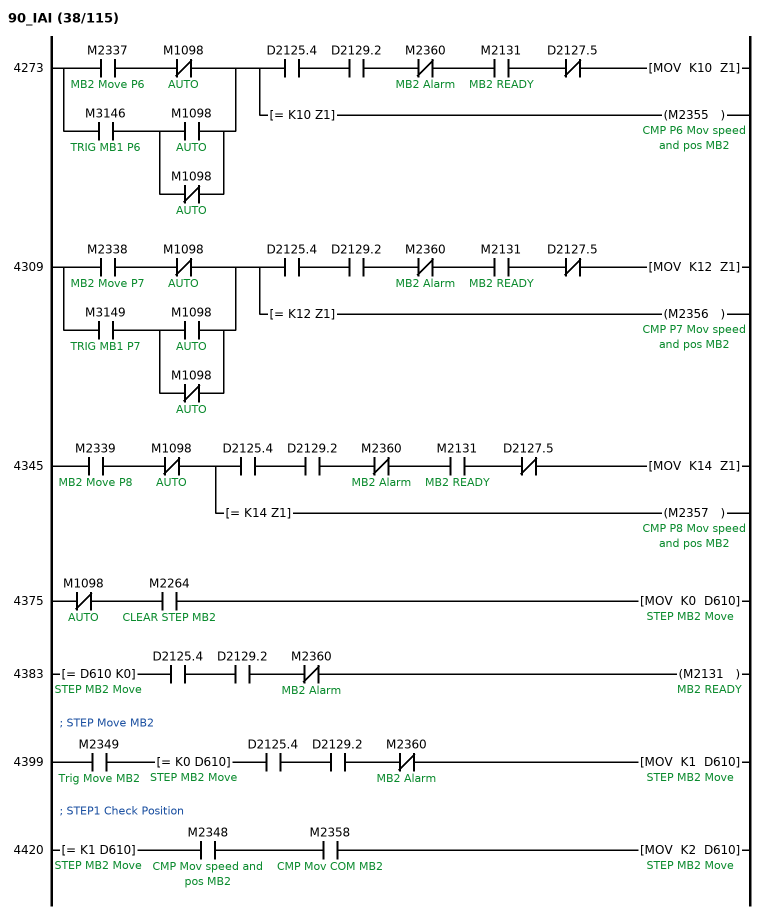
4273  LD      M2337  ; MB2 Move P6
      ANI     M1098  ; AUTO
      LD      M3146  ; TRIG MB1 P6
      LD      M1098  ; AUTO
      ORI     M1098  ; AUTO
      ANB
      ORB
      MPS
      AND     D2125.4
      AND     D2129.2
      ANI     M2360  ; MB2 Alarm
      AND     M2131  ; MB2 READY
      ANI     D2127.5
      MOV     K10 Z1
      MPP
      AND=    K10 Z1
      OUT     M2355  ; CMP P6 Mov speed and pos MB2
4309  LD      M2338  ; MB2 Move P7
      ANI     M1098  ; AUTO
      LD      M3149  ; TRIG MB1 P7
      LD      M1098  ; AUTO
      ORI     M1098  ; AUTO
      ANB
      ORB
      MPS
      AND     D2125.4
      AND     D2129.2
      ANI     M2360  ; MB2 Alarm
      AND     M2131  ; MB2 READY
      ANI     D2127.5
      MOV     K12 Z1
      MPP
      AND=    K12 Z1
      OUT     M2356  ; CMP P7 Mov speed and pos MB2
4345  LD      M2339  ; MB2 Move P8
      ANI     M1098  ; AUTO
      MPS
      AND     D2125.4
      AND     D2129.2
      ANI     M2360  ; MB2 Alarm
      AND     M2131  ; MB2 READY
      ANI     D2127.5
      MOV     K14 Z1
      MPP
      AND=    K14 Z1
      OUT     M2357  ; CMP P8 Mov speed and pos MB2
4375  LDI     M1098  ; AUTO
      AND     M2264  ; CLEAR STEP MB2
      MOV     K0 D610
4383  LD=     D610 K0  ; STEP MB2 Move
      AND     D2125.4
      AND     D2129.2
      ANI     M2360  ; MB2 Alarm
      OUT     M2131  ; MB2 READY
; STEP Move MB2
4399  LD      M2349  ; Trig Move MB2
      AND=    K0 D610  ; STEP MB2 Move
      AND     D2125.4
      AND     D2129.2
      ANI     M2360  ; MB2 Alarm
      MOV     K1 D610
; STEP1 Check Position
4420  LD=     K1 D610  ; STEP MB2 Move
      AND     M2348  ; CMP Mov speed and pos MB2
      AND     M2358  ; CMP Mov COM MB2
      MOV     K2 D610
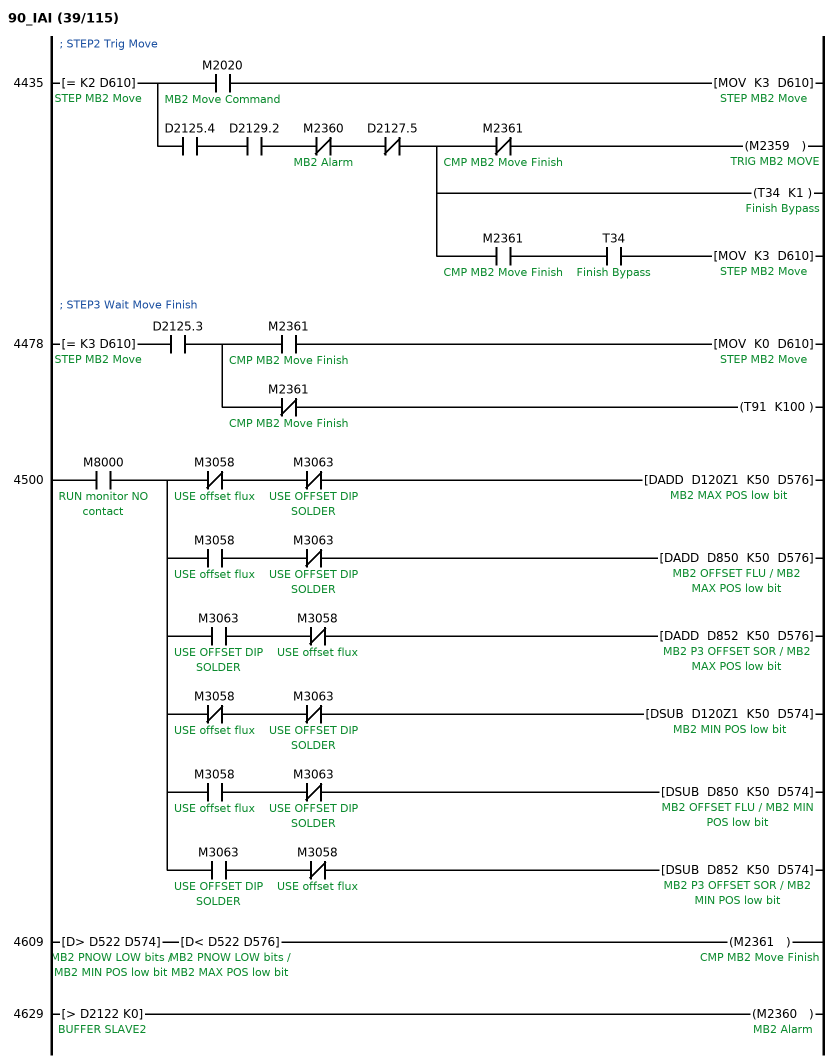
; STEP2 Trig Move
4435  LD=     K2 D610  ; STEP MB2 Move
      MPS
      AND     M2020  ; MB2 Move Command
      MOV     K3 D610
      MPP
      AND     D2125.4
      AND     D2129.2
      ANI     M2360  ; MB2 Alarm
      ANI     D2127.5
      MPS
      ANI     M2361  ; CMP MB2 Move Finish
      OUT     M2359  ; TRIG MB2 MOVE
      MPP
      OUT     T34 K1  ; Finish Bypass
      AND     M2361  ; CMP MB2 Move Finish
      AND     T34  ; Finish Bypass
      MOV     K3 D610
; STEP3 Wait Move Finish
4478  LD=     K3 D610  ; STEP MB2 Move
      AND     D2125.3
      MPS
      AND     M2361  ; CMP MB2 Move Finish
      MOV     K0 D610
      MPP
      ANI     M2361  ; CMP MB2 Move Finish
      OUT     T91 K100
4500  LD      M8000  ; RUN monitor NO contact
      MPS
      ANI     M3058  ; USE offset flux
      ANI     M3063  ; USE OFFSET DIP SOLDER
      DADD    D120Z1 K50 D576  ; MB2 MAX POS low bit
      MRD
      AND     M3058  ; USE offset flux
      ANI     M3063  ; USE OFFSET DIP SOLDER
      DADD    D850 K50 D576
      MRD
      AND     M3063  ; USE OFFSET DIP SOLDER
      ANI     M3058  ; USE offset flux
      DADD    D852 K50 D576
      MRD
      ANI     M3058  ; USE offset flux
      ANI     M3063  ; USE OFFSET DIP SOLDER
      DSUB    D120Z1 K50 D574  ; MB2 MIN POS low bit
      MRD
      AND     M3058  ; USE offset flux
      ANI     M3063  ; USE OFFSET DIP SOLDER
      DSUB    D850 K50 D574
      MPP
      AND     M3063  ; USE OFFSET DIP SOLDER
      ANI     M3058  ; USE offset flux
      DSUB    D852 K50 D574
4609  LDD>    D522 D574  ; MB2 PNOW LOW bits / MB2 MIN POS low bit
      ANDD<   D522 D576  ; MB2 PNOW LOW bits / MB2 MAX POS low bit
      OUT     M2361  ; CMP MB2 Move Finish
4629  LD>     D2122 K0  ; BUFFER SLAVE2
      OUT     M2360  ; MB2 Alarm
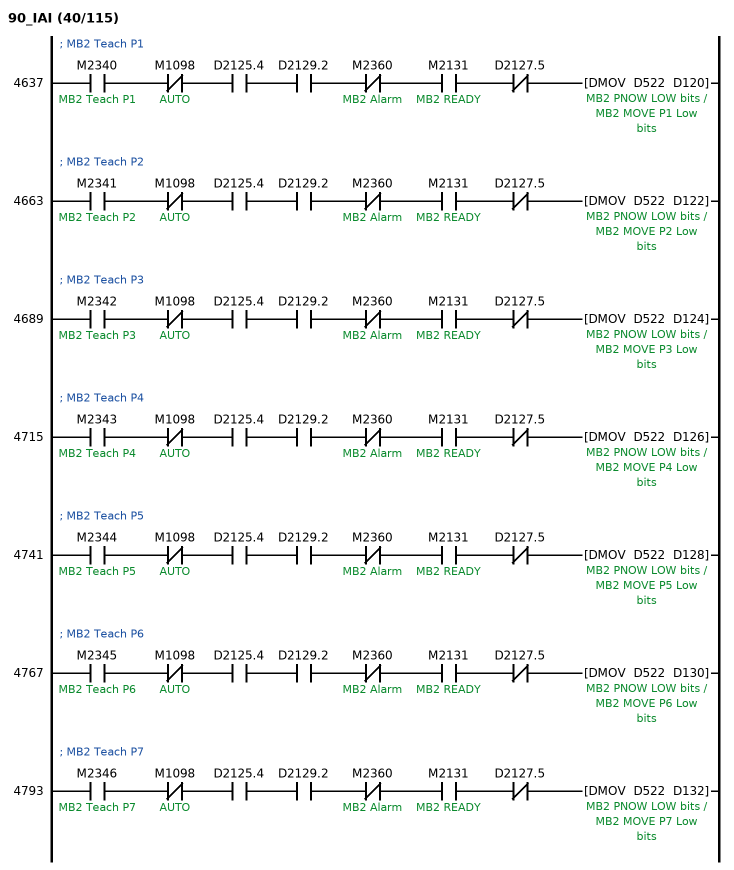
; MB2 Teach P1
4637  LD      M2340  ; MB2 Teach P1
      ANI     M1098  ; AUTO
      AND     D2125.4
      AND     D2129.2
      ANI     M2360  ; MB2 Alarm
      AND     M2131  ; MB2 READY
      ANI     D2127.5
      DMOV    D522 D120  ; MB2 MOVE P1 Low bits
; MB2 Teach P2
4663  LD      M2341  ; MB2 Teach P2
      ANI     M1098  ; AUTO
      AND     D2125.4
      AND     D2129.2
      ANI     M2360  ; MB2 Alarm
      AND     M2131  ; MB2 READY
      ANI     D2127.5
      DMOV    D522 D122  ; MB2 MOVE P2 Low bits
; MB2 Teach P3
4689  LD      M2342  ; MB2 Teach P3
      ANI     M1098  ; AUTO
      AND     D2125.4
      AND     D2129.2
      ANI     M2360  ; MB2 Alarm
      AND     M2131  ; MB2 READY
      ANI     D2127.5
      DMOV    D522 D124  ; MB2 MOVE P3 Low bits
; MB2 Teach P4
4715  LD      M2343  ; MB2 Teach P4
      ANI     M1098  ; AUTO
      AND     D2125.4
      AND     D2129.2
      ANI     M2360  ; MB2 Alarm
      AND     M2131  ; MB2 READY
      ANI     D2127.5
      DMOV    D522 D126  ; MB2 MOVE P4 Low bits
; MB2 Teach P5
4741  LD      M2344  ; MB2 Teach P5
      ANI     M1098  ; AUTO
      AND     D2125.4
      AND     D2129.2
      ANI     M2360  ; MB2 Alarm
      AND     M2131  ; MB2 READY
      ANI     D2127.5
      DMOV    D522 D128  ; MB2 MOVE P5 Low bits
; MB2 Teach P6
4767  LD      M2345  ; MB2 Teach P6
      ANI     M1098  ; AUTO
      AND     D2125.4
      AND     D2129.2
      ANI     M2360  ; MB2 Alarm
      AND     M2131  ; MB2 READY
      ANI     D2127.5
      DMOV    D522 D130  ; MB2 MOVE P6 Low bits
; MB2 Teach P7
4793  LD      M2346  ; MB2 Teach P7
      ANI     M1098  ; AUTO
      AND     D2125.4
      AND     D2129.2
      ANI     M2360  ; MB2 Alarm
      AND     M2131  ; MB2 READY
      ANI     D2127.5
      DMOV    D522 D132  ; MB2 MOVE P7 Low bits
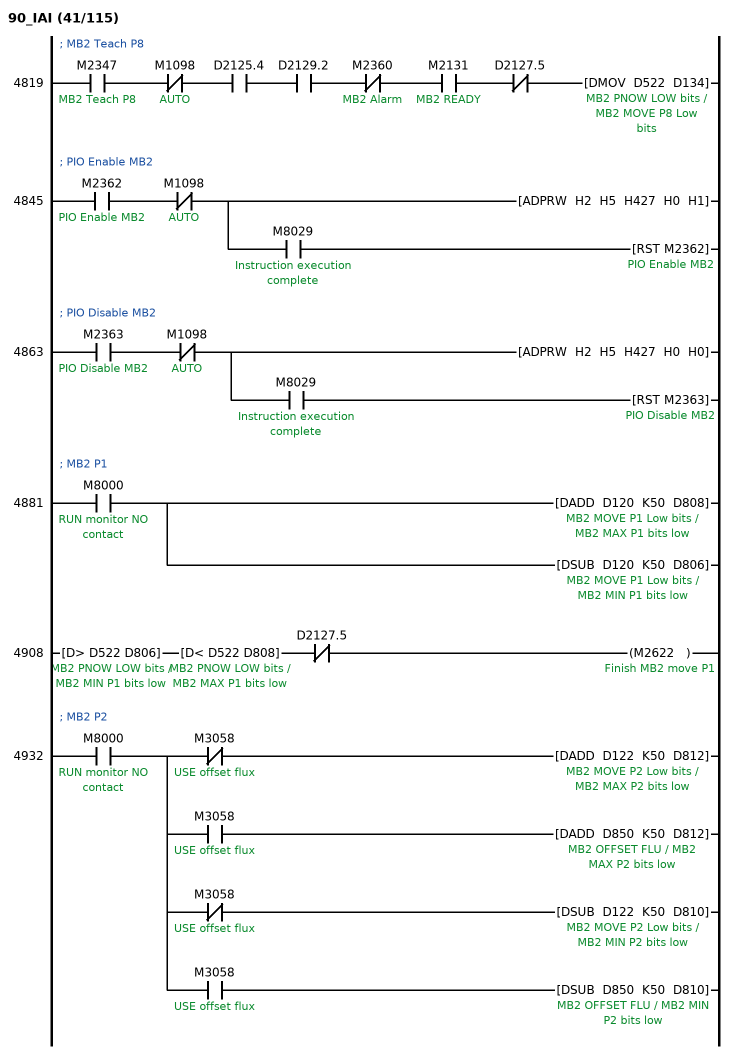
; MB2 Teach P8
4819  LD      M2347  ; MB2 Teach P8
      ANI     M1098  ; AUTO
      AND     D2125.4
      AND     D2129.2
      ANI     M2360  ; MB2 Alarm
      AND     M2131  ; MB2 READY
      ANI     D2127.5
      DMOV    D522 D134  ; MB2 MOVE P8 Low bits
; PIO Enable MB2
4845  LD      M2362  ; PIO Enable MB2
      ANI     M1098  ; AUTO
      ADPRW   H2 H5 H427 H0 H1
      AND     M8029  ; Instruction execution complete
      RST     M2362  ; PIO Enable MB2
; PIO Disable MB2
4863  LD      M2363  ; PIO Disable MB2
      ANI     M1098  ; AUTO
      ADPRW   H2 H5 H427 H0 H0
      AND     M8029  ; Instruction execution complete
      RST     M2363  ; PIO Disable MB2
; MB2 P1
4881  LD      M8000  ; RUN monitor NO contact
      DADD    D120 K50 D808  ; MB2 MAX P1 bits low
      DSUB    D120 K50 D806  ; MB2 MIN P1 bits low
4908  LDD>    D522 D806  ; MB2 PNOW LOW bits / MB2 MIN P1 bits low
      ANDD<   D522 D808  ; MB2 PNOW LOW bits / MB2 MAX P1 bits low
      ANI     D2127.5
      OUT     M2622  ; Finish MB2 move P1
; MB2 P2
4932  LD      M8000  ; RUN monitor NO contact
      MPS
      ANI     M3058  ; USE offset flux
      DADD    D122 K50 D812  ; MB2 MAX P2 bits low
      MRD
      AND     M3058  ; USE offset flux
      DADD    D850 K50 D812
      MRD
      ANI     M3058  ; USE offset flux
      DSUB    D122 K50 D810  ; MB2 MIN P2 bits low
      MPP
      AND     M3058  ; USE offset flux
      DSUB    D850 K50 D810
